// TIA Portal V17 export
// export: Created 2025-03-05T08:00:11.0156381Z, ExportSetting WithDefaults, DisplayName Totally Integrated Automation Portal, DisplayVersion V17 Update 8, DisplayName TIA Portal Openness, DisplayVersion V17 Update 8, DisplayName TIA Portal Version Control Interface, DisplayVersion V17, DisplayName SINAMICS Startdrive Advanced, DisplayVersion V17 SP2, DisplayName SINAMICS Startdrive G110M, G120, G120C, G120D, G120P, G115D, DisplayVersion V17 SP2, DisplayName SINAMICS Startdrive G130, G150, S120, S150, SINAMICS MV, S210, DisplayVersion V17 SP2, DisplayName STEP 7 Professional, DisplayVersion V17 Update 8, DisplayName SINUMERIK ONE STEP 7 Toolbox, DisplayVersion V17 Update 12, DisplayName SINUMERIK 840D sl STEP 7 Toolbox, DisplayVersion V17 Update 12, DisplayName STEP 7 Safety, DisplayVersion V17 Update 6, DisplayName WinCC Advanced, DisplayVersion V17 Update 8
FUNCTION "FC2122_HT10" : Void   // FC2122, LAD
{ S7_Optimized_Access := 'TRUE' }
AUTHOR : ETXETAR
VERSION : 1.0
// stored: AutoNumber false, IsIECCheckEnabled false, SetENOAutomatically false, UDAEnableTagReadback false
   VAR CONSTANT
      FC_NUMBER : DInt := 2122;   // FC NUMEBR
   END_VAR
   VAR_TEMP   // added for the SCL form of the ladder/FBD networks
      _w1 : Bool;
      _w2 : Bool;
      _w3 : Bool;
   END_VAR
BEGIN

REGION Network 1: INPUT HT10 EMERGENCY STOP
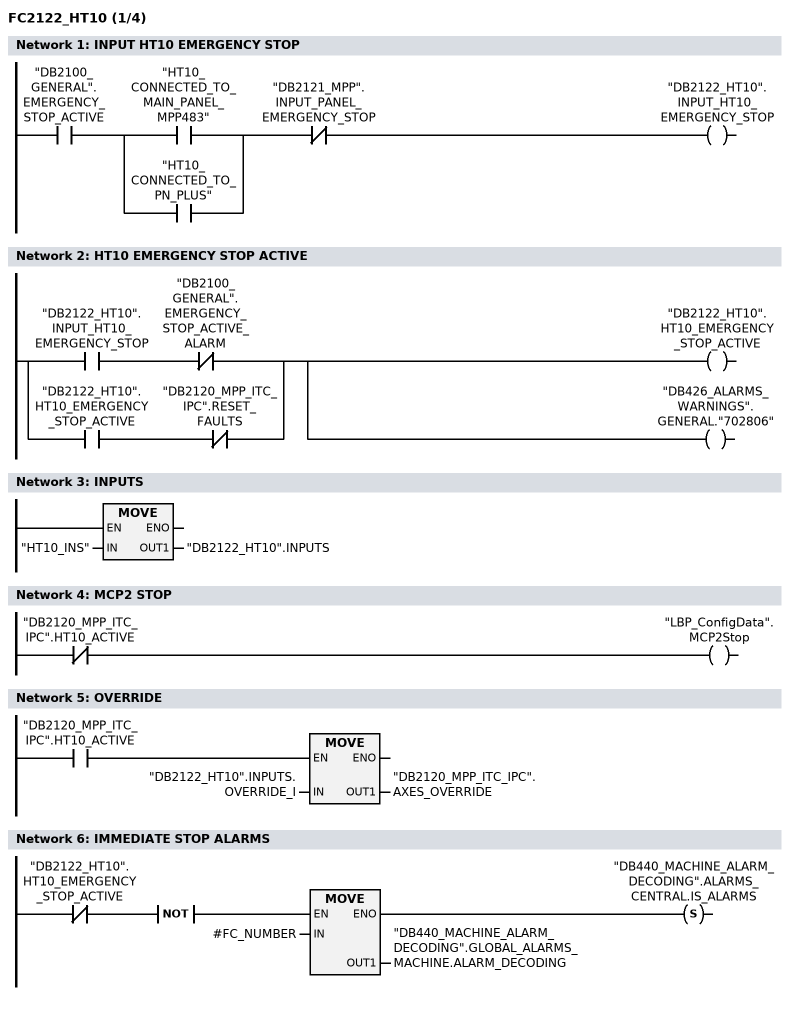
   RUNG wire#powerrail
      Contact( "DB2100_GENERAL".EMERGENCY_STOP_ACTIVE )
      wire#w1
      Contact( "HT10_CONNECTED_TO_MAIN_PANEL_MPP483" )
      wire#w2
      I_Contact( "DB2121_MPP".INPUT_PANEL_EMERGENCY_STOP )
      Coil( "DB2122_HT10".INPUT_HT10_EMERGENCY_STOP )
   END_RUNG
   RUNG wire#w1
      Contact( "HT10_CONNECTED_TO_PN_PLUS" )
   END_RUNG wire#w2
   // the same network as SCL:
   "DB2122_HT10".INPUT_HT10_EMERGENCY_STOP := "DB2100_GENERAL".EMERGENCY_STOP_ACTIVE AND ("HT10_CONNECTED_TO_MAIN_PANEL_MPP483" OR "HT10_CONNECTED_TO_PN_PLUS") AND NOT "DB2121_MPP".INPUT_PANEL_EMERGENCY_STOP;
END_REGION

REGION Network 2: HT10 EMERGENCY STOP ACTIVE
   RUNG wire#powerrail
      Contact( "DB2122_HT10".INPUT_HT10_EMERGENCY_STOP )
      I_Contact( "DB2100_GENERAL".EMERGENCY_STOP_ACTIVE_ALARM )
      wire#w1
      Coil( "DB2122_HT10".HT10_EMERGENCY_STOP_ACTIVE )
   END_RUNG
   RUNG wire#powerrail
      Contact( "DB2122_HT10".HT10_EMERGENCY_STOP_ACTIVE )
      I_Contact( "DB2120_MPP_ITC_IPC".RESET_FAULTS )
   END_RUNG wire#w1
   RUNG wire#w1
      Coil( "DB426_ALARMS_WARNINGS".GENERAL."702806" )
   END_RUNG
   // the same network as SCL:
   "DB2122_HT10".HT10_EMERGENCY_STOP_ACTIVE := ("DB2122_HT10".INPUT_HT10_EMERGENCY_STOP AND NOT "DB2100_GENERAL".EMERGENCY_STOP_ACTIVE_ALARM) OR ("DB2122_HT10".HT10_EMERGENCY_STOP_ACTIVE AND NOT "DB2120_MPP_ITC_IPC".RESET_FAULTS);
   "DB426_ALARMS_WARNINGS".GENERAL."702806" := "DB2122_HT10".HT10_EMERGENCY_STOP_ACTIVE;
END_REGION

REGION Network 3: INPUTS
   RUNG wire#powerrail
      Move(in := "HT10_INS", out1 => "DB2122_HT10".INPUTS)
   END_RUNG
   // the same network as SCL:
   "DB2122_HT10".INPUTS := "HT10_INS";
END_REGION

REGION Network 4: MCP2 STOP
   RUNG wire#powerrail
      I_Contact( "DB2120_MPP_ITC_IPC".HT10_ACTIVE )
      Coil( "LBP_ConfigData".MCP2Stop )
   END_RUNG
   // the same network as SCL:
   "LBP_ConfigData".MCP2Stop := NOT "DB2120_MPP_ITC_IPC".HT10_ACTIVE;
END_REGION

REGION Network 5: OVERRIDE
   RUNG wire#powerrail
      Contact( "DB2120_MPP_ITC_IPC".HT10_ACTIVE )
      Move(in := "DB2122_HT10".INPUTS.OVERRIDE_I, out1 => "DB2120_MPP_ITC_IPC".AXES_OVERRIDE)
   END_RUNG
   // the same network as SCL:
   IF "DB2120_MPP_ITC_IPC".HT10_ACTIVE THEN
       "DB2120_MPP_ITC_IPC".AXES_OVERRIDE := "DB2122_HT10".INPUTS.OVERRIDE_I;
   END_IF;
END_REGION

REGION Network 6: IMMEDIATE STOP ALARMS
   RUNG wire#powerrail
      I_Contact( "DB2122_HT10".HT10_EMERGENCY_STOP_ACTIVE )
      Not()
      { S7_GenerateENO := "TRUE" } Move(in := #FC_NUMBER, out1 => "DB440_MACHINE_ALARM_DECODING".GLOBAL_ALARMS_MACHINE.ALARM_DECODING)
      S_Coil( "DB440_MACHINE_ALARM_DECODING".ALARMS_CENTRAL.IS_ALARMS )
   END_RUNG
   // the same network as SCL:
   // ENO of a box is taken as its EN; it also drops when the box reports an error
   IF NOT (NOT "DB2122_HT10".HT10_EMERGENCY_STOP_ACTIVE) THEN
       "DB440_MACHINE_ALARM_DECODING".GLOBAL_ALARMS_MACHINE.ALARM_DECODING := #FC_NUMBER;
       "DB440_MACHINE_ALARM_DECODING".ALARMS_CENTRAL.IS_ALARMS := TRUE;
   END_IF;
END_REGION

REGION Network 7: OUTPUTS
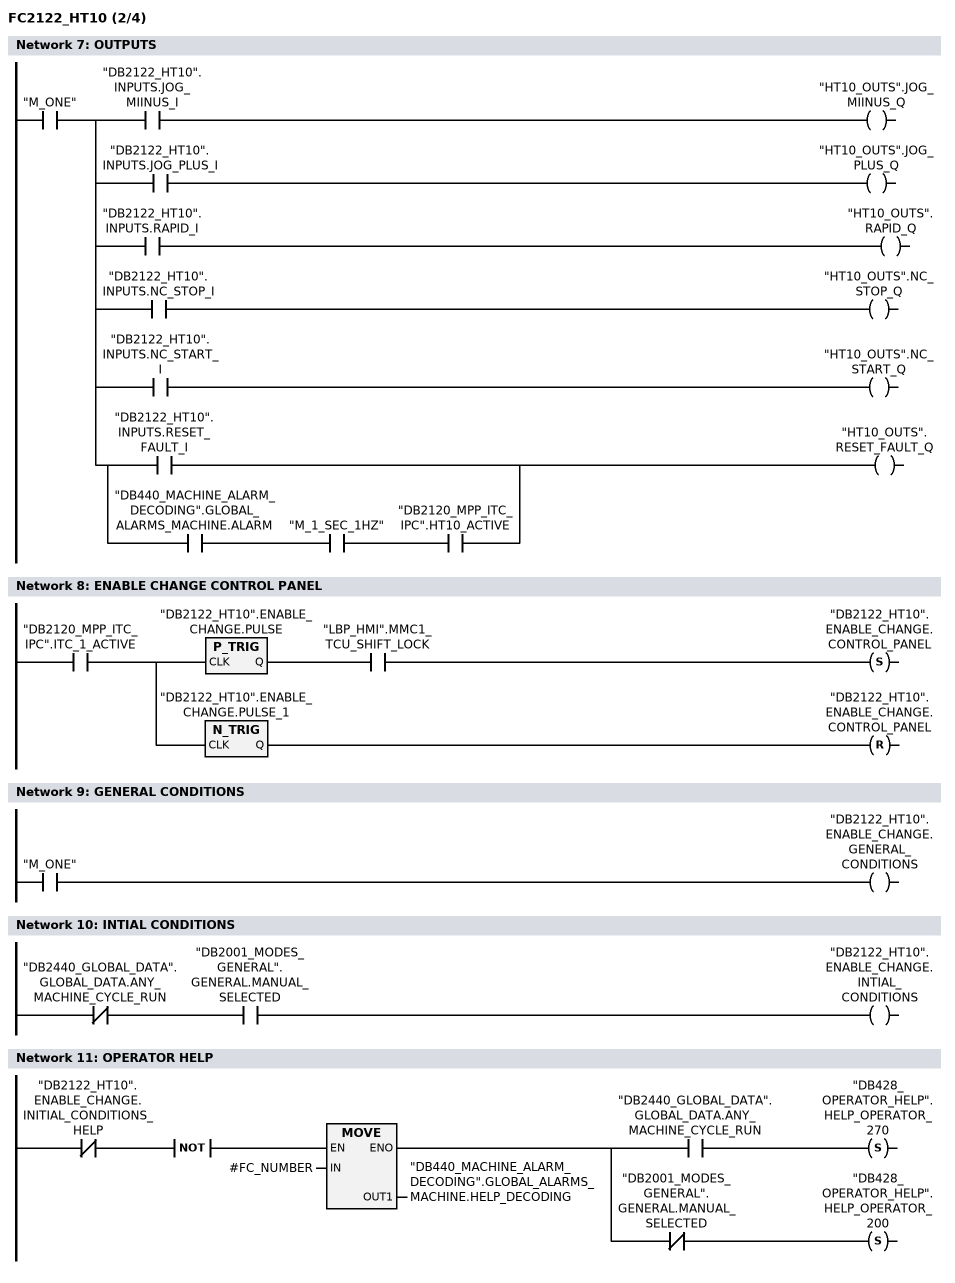
   RUNG wire#powerrail
      Contact( "M_ONE" )
      wire#w1
      Contact( "DB2122_HT10".INPUTS.JOG_MIINUS_I )
      Coil( "HT10_OUTS".JOG_MIINUS_Q )
   END_RUNG
   RUNG wire#w1
      Contact( "DB2122_HT10".INPUTS.JOG_PLUS_I )
      Coil( "HT10_OUTS".JOG_PLUS_Q )
   END_RUNG
   RUNG wire#w1
      Contact( "DB2122_HT10".INPUTS.RAPID_I )
      Coil( "HT10_OUTS".RAPID_Q )
   END_RUNG
   RUNG wire#w1
      Contact( "DB2122_HT10".INPUTS.NC_STOP_I )
      Coil( "HT10_OUTS".NC_STOP_Q )
   END_RUNG
   RUNG wire#w1
      Contact( "DB2122_HT10".INPUTS.NC_START_I )
      Coil( "HT10_OUTS".NC_START_Q )
   END_RUNG
   RUNG wire#w1
      Contact( "DB2122_HT10".INPUTS.RESET_FAULT_I )
      wire#w2
      Coil( "HT10_OUTS".RESET_FAULT_Q )
   END_RUNG
   RUNG wire#w1
      Contact( "DB440_MACHINE_ALARM_DECODING".GLOBAL_ALARMS_MACHINE.ALARM )
      Contact( "M_1_SEC_1HZ" )
      Contact( "DB2120_MPP_ITC_IPC".HT10_ACTIVE )
   END_RUNG wire#w2
   // the same network as SCL:
   "HT10_OUTS".JOG_MIINUS_Q := "M_ONE" AND "DB2122_HT10".INPUTS.JOG_MIINUS_I;
   "HT10_OUTS".JOG_PLUS_Q := "M_ONE" AND "DB2122_HT10".INPUTS.JOG_PLUS_I;
   "HT10_OUTS".RAPID_Q := "M_ONE" AND "DB2122_HT10".INPUTS.RAPID_I;
   "HT10_OUTS".NC_STOP_Q := "M_ONE" AND "DB2122_HT10".INPUTS.NC_STOP_I;
   "HT10_OUTS".NC_START_Q := "M_ONE" AND "DB2122_HT10".INPUTS.NC_START_I;
   "HT10_OUTS".RESET_FAULT_Q := "M_ONE" AND ("DB2122_HT10".INPUTS.RESET_FAULT_I OR ("DB440_MACHINE_ALARM_DECODING".GLOBAL_ALARMS_MACHINE.ALARM AND "M_1_SEC_1HZ" AND "DB2120_MPP_ITC_IPC".HT10_ACTIVE));
END_REGION

REGION Network 8: ENABLE CHANGE CONTROL PANEL
   RUNG wire#powerrail
      Contact( "DB2120_MPP_ITC_IPC".ITC_1_ACTIVE )
      wire#w1
      P_Trig( "DB2122_HT10".ENABLE_CHANGE.PULSE )
      Contact( "LBP_HMI".MMC1_TCU_SHIFT_LOCK )
      S_Coil( "DB2122_HT10".ENABLE_CHANGE.CONTROL_PANEL )
   END_RUNG
   RUNG wire#w1
      N_Trig( "DB2122_HT10".ENABLE_CHANGE.PULSE_1 )
      R_Coil( "DB2122_HT10".ENABLE_CHANGE.CONTROL_PANEL )
   END_RUNG
   // the same network as SCL:
   #_w1 := "DB2120_MPP_ITC_IPC".ITC_1_ACTIVE AND NOT "DB2122_HT10".ENABLE_CHANGE.PULSE;   // rising edge
   "DB2122_HT10".ENABLE_CHANGE.PULSE := "DB2120_MPP_ITC_IPC".ITC_1_ACTIVE;
   IF #_w1 AND "LBP_HMI".MMC1_TCU_SHIFT_LOCK THEN "DB2122_HT10".ENABLE_CHANGE.CONTROL_PANEL := TRUE; END_IF;
   #_w2 := NOT "DB2120_MPP_ITC_IPC".ITC_1_ACTIVE AND "DB2122_HT10".ENABLE_CHANGE.PULSE_1;   // falling edge
   "DB2122_HT10".ENABLE_CHANGE.PULSE_1 := "DB2120_MPP_ITC_IPC".ITC_1_ACTIVE;
   IF #_w2 THEN "DB2122_HT10".ENABLE_CHANGE.CONTROL_PANEL := FALSE; END_IF;
END_REGION

REGION Network 9: GENERAL CONDITIONS
   RUNG wire#powerrail
      Contact( "M_ONE" )
      Coil( "DB2122_HT10".ENABLE_CHANGE.GENERAL_CONDITIONS )
   END_RUNG
   // the same network as SCL:
   "DB2122_HT10".ENABLE_CHANGE.GENERAL_CONDITIONS := "M_ONE";
END_REGION

REGION Network 10: INTIAL CONDITIONS
   RUNG wire#powerrail
      I_Contact( "DB2440_GLOBAL_DATA".GLOBAL_DATA.ANY_MACHINE_CYCLE_RUN )
      Contact( "DB2001_MODES_GENERAL".GENERAL.MANUAL_SELECTED )
      Coil( "DB2122_HT10".ENABLE_CHANGE.INTIAL_CONDITIONS )
   END_RUNG
   // the same network as SCL:
   "DB2122_HT10".ENABLE_CHANGE.INTIAL_CONDITIONS := NOT "DB2440_GLOBAL_DATA".GLOBAL_DATA.ANY_MACHINE_CYCLE_RUN AND "DB2001_MODES_GENERAL".GENERAL.MANUAL_SELECTED;
END_REGION

REGION Network 11: OPERATOR HELP
   RUNG wire#powerrail
      I_Contact( "DB2122_HT10".ENABLE_CHANGE.INITIAL_CONDITIONS_HELP )
      Not()
      { S7_GenerateENO := "TRUE" } Move(in := #FC_NUMBER, out1 => "DB440_MACHINE_ALARM_DECODING".GLOBAL_ALARMS_MACHINE.HELP_DECODING)
      wire#w1
      Contact( "DB2440_GLOBAL_DATA".GLOBAL_DATA.ANY_MACHINE_CYCLE_RUN )
      S_Coil( "DB428_OPERATOR_HELP".HELP_OPERATOR_270 )
   END_RUNG
   RUNG wire#w1
      I_Contact( "DB2001_MODES_GENERAL".GENERAL.MANUAL_SELECTED )
      S_Coil( "DB428_OPERATOR_HELP".HELP_OPERATOR_200 )
   END_RUNG
   // the same network as SCL:
   // ENO of a box is taken as its EN; it also drops when the box reports an error
   #_w1 := NOT (NOT "DB2122_HT10".ENABLE_CHANGE.INITIAL_CONDITIONS_HELP);
   IF #_w1 THEN "DB440_MACHINE_ALARM_DECODING".GLOBAL_ALARMS_MACHINE.HELP_DECODING := #FC_NUMBER; END_IF;
   IF #_w1 AND "DB2440_GLOBAL_DATA".GLOBAL_DATA.ANY_MACHINE_CYCLE_RUN THEN
       "DB428_OPERATOR_HELP".HELP_OPERATOR_270 := TRUE;
   END_IF;
   IF #_w1 AND NOT "DB2001_MODES_GENERAL".GENERAL.MANUAL_SELECTED THEN
       "DB428_OPERATOR_HELP".HELP_OPERATOR_200 := TRUE;
   END_IF;
END_REGION

REGION Network 12: MANUAL REQUEST
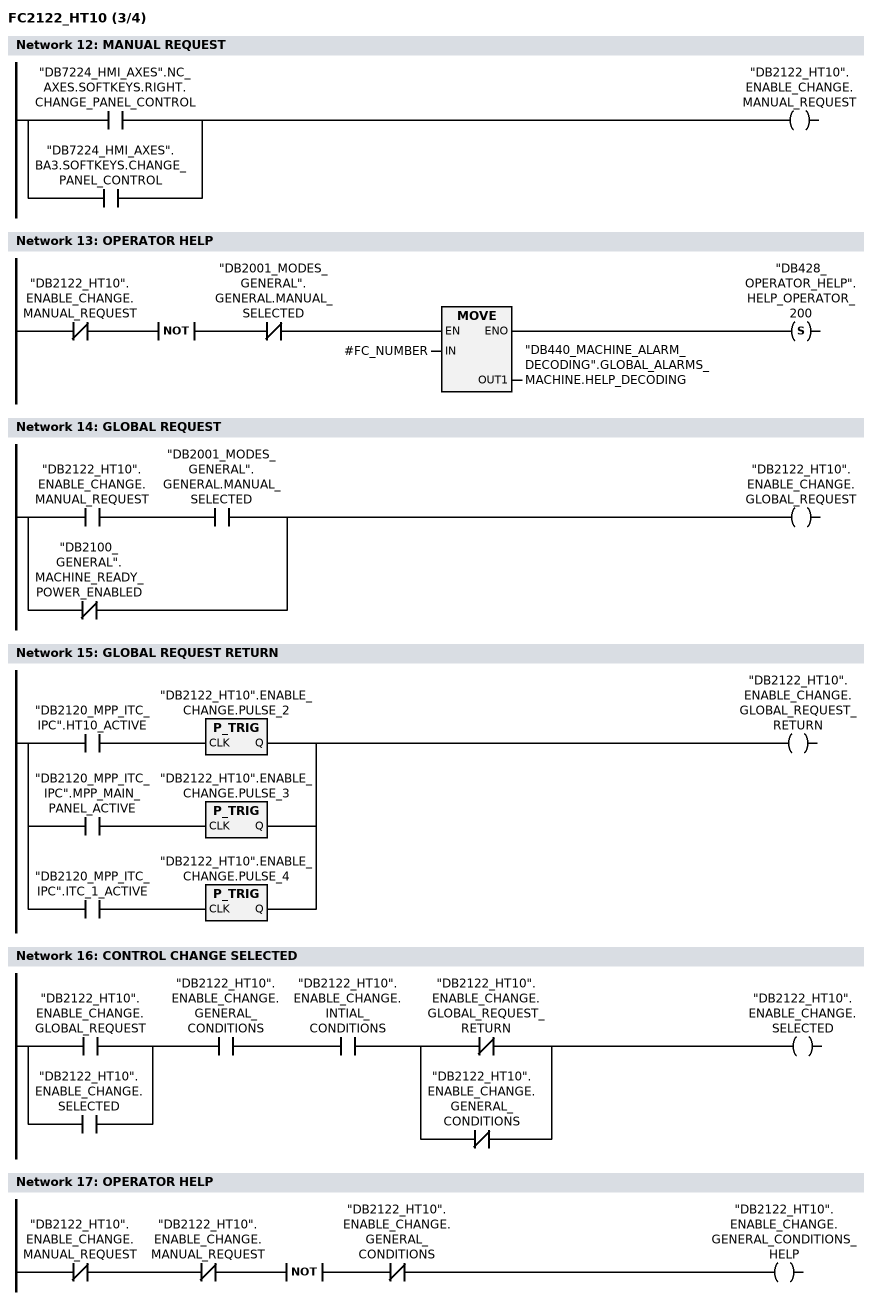
   RUNG wire#powerrail
      Contact( "DB7224_HMI_AXES".NC_AXES.SOFTKEYS.RIGHT.CHANGE_PANEL_CONTROL )
      wire#w1
      Coil( "DB2122_HT10".ENABLE_CHANGE.MANUAL_REQUEST )
   END_RUNG
   RUNG wire#powerrail
      Contact( "DB7224_HMI_AXES".BA3.SOFTKEYS.CHANGE_PANEL_CONTROL )
   END_RUNG wire#w1
   // the same network as SCL:
   "DB2122_HT10".ENABLE_CHANGE.MANUAL_REQUEST := "DB7224_HMI_AXES".NC_AXES.SOFTKEYS.RIGHT.CHANGE_PANEL_CONTROL OR "DB7224_HMI_AXES".BA3.SOFTKEYS.CHANGE_PANEL_CONTROL;
END_REGION

REGION Network 13: OPERATOR HELP
   RUNG wire#powerrail
      I_Contact( "DB2122_HT10".ENABLE_CHANGE.MANUAL_REQUEST )
      Not()
      I_Contact( "DB2001_MODES_GENERAL".GENERAL.MANUAL_SELECTED )
      { S7_GenerateENO := "TRUE" } Move(in := #FC_NUMBER, out1 => "DB440_MACHINE_ALARM_DECODING".GLOBAL_ALARMS_MACHINE.HELP_DECODING)
      S_Coil( "DB428_OPERATOR_HELP".HELP_OPERATOR_200 )
   END_RUNG
   // the same network as SCL:
   // ENO of a box is taken as its EN; it also drops when the box reports an error
   IF NOT (NOT "DB2122_HT10".ENABLE_CHANGE.MANUAL_REQUEST) AND NOT "DB2001_MODES_GENERAL".GENERAL.MANUAL_SELECTED THEN
       "DB440_MACHINE_ALARM_DECODING".GLOBAL_ALARMS_MACHINE.HELP_DECODING := #FC_NUMBER;
       "DB428_OPERATOR_HELP".HELP_OPERATOR_200 := TRUE;
   END_IF;
END_REGION

REGION Network 14: GLOBAL REQUEST
   RUNG wire#powerrail
      Contact( "DB2122_HT10".ENABLE_CHANGE.MANUAL_REQUEST )
      Contact( "DB2001_MODES_GENERAL".GENERAL.MANUAL_SELECTED )
      wire#w1
      Coil( "DB2122_HT10".ENABLE_CHANGE.GLOBAL_REQUEST )
   END_RUNG
   RUNG wire#powerrail
      I_Contact( "DB2100_GENERAL".MACHINE_READY_POWER_ENABLED )
   END_RUNG wire#w1
   // the same network as SCL:
   "DB2122_HT10".ENABLE_CHANGE.GLOBAL_REQUEST := ("DB2122_HT10".ENABLE_CHANGE.MANUAL_REQUEST AND "DB2001_MODES_GENERAL".GENERAL.MANUAL_SELECTED) OR NOT "DB2100_GENERAL".MACHINE_READY_POWER_ENABLED;
END_REGION

REGION Network 15: GLOBAL REQUEST RETURN
   RUNG wire#powerrail
      Contact( "DB2120_MPP_ITC_IPC".HT10_ACTIVE )
      P_Trig( "DB2122_HT10".ENABLE_CHANGE.PULSE_2 )
      wire#w1
      Coil( "DB2122_HT10".ENABLE_CHANGE.GLOBAL_REQUEST_RETURN )
   END_RUNG
   RUNG wire#powerrail
      Contact( "DB2120_MPP_ITC_IPC".MPP_MAIN_PANEL_ACTIVE )
      P_Trig( "DB2122_HT10".ENABLE_CHANGE.PULSE_3 )
   END_RUNG wire#w1
   RUNG wire#powerrail
      Contact( "DB2120_MPP_ITC_IPC".ITC_1_ACTIVE )
      P_Trig( "DB2122_HT10".ENABLE_CHANGE.PULSE_4 )
   END_RUNG wire#w1
   // the same network as SCL:
   #_w1 := "DB2120_MPP_ITC_IPC".HT10_ACTIVE AND NOT "DB2122_HT10".ENABLE_CHANGE.PULSE_2;   // rising edge
   "DB2122_HT10".ENABLE_CHANGE.PULSE_2 := "DB2120_MPP_ITC_IPC".HT10_ACTIVE;
   #_w2 := "DB2120_MPP_ITC_IPC".MPP_MAIN_PANEL_ACTIVE AND NOT "DB2122_HT10".ENABLE_CHANGE.PULSE_3;   // rising edge
   "DB2122_HT10".ENABLE_CHANGE.PULSE_3 := "DB2120_MPP_ITC_IPC".MPP_MAIN_PANEL_ACTIVE;
   #_w3 := "DB2120_MPP_ITC_IPC".ITC_1_ACTIVE AND NOT "DB2122_HT10".ENABLE_CHANGE.PULSE_4;   // rising edge
   "DB2122_HT10".ENABLE_CHANGE.PULSE_4 := "DB2120_MPP_ITC_IPC".ITC_1_ACTIVE;
   "DB2122_HT10".ENABLE_CHANGE.GLOBAL_REQUEST_RETURN := #_w1 OR #_w2 OR #_w3;
END_REGION

REGION Network 16: CONTROL CHANGE SELECTED
   RUNG wire#powerrail
      Contact( "DB2122_HT10".ENABLE_CHANGE.GLOBAL_REQUEST )
      wire#w1
      Contact( "DB2122_HT10".ENABLE_CHANGE.GENERAL_CONDITIONS )
      Contact( "DB2122_HT10".ENABLE_CHANGE.INTIAL_CONDITIONS )
      wire#w2
      I_Contact( "DB2122_HT10".ENABLE_CHANGE.GLOBAL_REQUEST_RETURN )
      wire#w3
      Coil( "DB2122_HT10".ENABLE_CHANGE.SELECTED )
   END_RUNG
   RUNG wire#powerrail
      Contact( "DB2122_HT10".ENABLE_CHANGE.SELECTED )
   END_RUNG wire#w1
   RUNG wire#w2
      I_Contact( "DB2122_HT10".ENABLE_CHANGE.GENERAL_CONDITIONS )
   END_RUNG wire#w3
   // the same network as SCL:
   "DB2122_HT10".ENABLE_CHANGE.SELECTED := ("DB2122_HT10".ENABLE_CHANGE.GLOBAL_REQUEST OR "DB2122_HT10".ENABLE_CHANGE.SELECTED) AND "DB2122_HT10".ENABLE_CHANGE.GENERAL_CONDITIONS AND "DB2122_HT10".ENABLE_CHANGE.INTIAL_CONDITIONS AND (NOT "DB2122_HT10".ENABLE_CHANGE.GLOBAL_REQUEST_RETURN OR NOT "DB2122_HT10".ENABLE_CHANGE.GENERAL_CONDITIONS);
END_REGION

REGION Network 17: OPERATOR HELP
   RUNG wire#powerrail
      I_Contact( "DB2122_HT10".ENABLE_CHANGE.MANUAL_REQUEST )
      I_Contact( "DB2122_HT10".ENABLE_CHANGE.MANUAL_REQUEST )
      Not()
      I_Contact( "DB2122_HT10".ENABLE_CHANGE.GENERAL_CONDITIONS )
      Coil( "DB2122_HT10".ENABLE_CHANGE.GENERAL_CONDITIONS_HELP )
   END_RUNG
   // the same network as SCL:
   "DB2122_HT10".ENABLE_CHANGE.GENERAL_CONDITIONS_HELP := NOT (NOT "DB2122_HT10".ENABLE_CHANGE.MANUAL_REQUEST AND NOT "DB2122_HT10".ENABLE_CHANGE.MANUAL_REQUEST) AND NOT "DB2122_HT10".ENABLE_CHANGE.GENERAL_CONDITIONS;
END_REGION

REGION Network 18: OPERATOR HELP
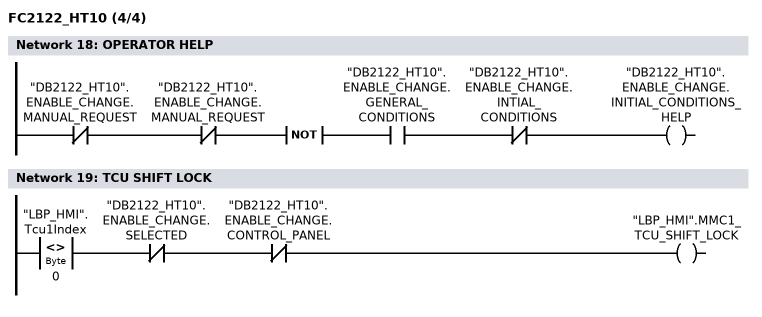
   RUNG wire#powerrail
      I_Contact( "DB2122_HT10".ENABLE_CHANGE.MANUAL_REQUEST )
      I_Contact( "DB2122_HT10".ENABLE_CHANGE.MANUAL_REQUEST )
      Not()
      Contact( "DB2122_HT10".ENABLE_CHANGE.GENERAL_CONDITIONS )
      I_Contact( "DB2122_HT10".ENABLE_CHANGE.INTIAL_CONDITIONS )
      Coil( "DB2122_HT10".ENABLE_CHANGE.INITIAL_CONDITIONS_HELP )
   END_RUNG
   // the same network as SCL:
   "DB2122_HT10".ENABLE_CHANGE.INITIAL_CONDITIONS_HELP := NOT (NOT "DB2122_HT10".ENABLE_CHANGE.MANUAL_REQUEST AND NOT "DB2122_HT10".ENABLE_CHANGE.MANUAL_REQUEST) AND "DB2122_HT10".ENABLE_CHANGE.GENERAL_CONDITIONS AND NOT "DB2122_HT10".ENABLE_CHANGE.INTIAL_CONDITIONS;
END_REGION

REGION Network 19: TCU SHIFT LOCK
   RUNG wire#powerrail
      { S7_Templates := "SrcType := Byte" } NE_Contact(in1 := "LBP_HMI".Tcu1Index, in2 := 0)
      I_Contact( "DB2122_HT10".ENABLE_CHANGE.SELECTED )
      I_Contact( "DB2122_HT10".ENABLE_CHANGE.CONTROL_PANEL )
      Coil( "LBP_HMI".MMC1_TCU_SHIFT_LOCK )
   END_RUNG
   // the same network as SCL:
   "LBP_HMI".MMC1_TCU_SHIFT_LOCK := ("LBP_HMI".Tcu1Index <> 0) AND NOT "DB2122_HT10".ENABLE_CHANGE.SELECTED AND NOT "DB2122_HT10".ENABLE_CHANGE.CONTROL_PANEL;
END_REGION
END_FUNCTION
